// TwinCAT 3 PLC project EnOcean
// ProgramVersion: 3.1.4022.4
// libraries:
//   Tc2_BABasic, * (Beckhoff Automation GmbH)
//   Tc2_EnOcean, * (Beckhoff Automation GmbH)
//   Tc2_Standard, * (Beckhoff Automation GmbH)
//   Tc2_System, * (Beckhoff Automation GmbH)
//   Tc2_Utilities, * (Beckhoff Automation GmbH)
//   Tc3_IotBase, * (Beckhoff Automation GmbH)
//   Tc3_Module, * (Beckhoff Automation GmbH)
// project tree:
//   / GlobalTextList.TcGTLO (not stored), PlcTask.TcTTO, Visualization Manager.TcVMO (not stored)
//   GVLs/ GVL_EnOcean.TcGVL, Waardes.TcGVL
//   POUs/FB/ didSensorChange.TcPOU, isOpen.TcPOU, readTemp2.TcPOU, switch2.TcPOU, contact2.TcPOU (not stored)
//   POUs/ JSonEncode.TcPOU, Main.TcPOU, mqttconn.TcPOU, readTemp.TcPOU, switch.TcPOU, contact.TcPOU (not stored)
//   VISUs/ Visualization.TcVIS (not stored)
// real-time tasks:
//   TASK PlcTask: cycle T#5ms, priority 15, ADS port 350
// I/O:
//   DEVICE Device 1 (EtherCAT) (disabled), AmsNetId 192.168.1.6.2.1
//     Term 1 (EK1200) [EK1200-5000 EtherCAT Power supply (2A E-Bus)]
//       Term 2 (EL1008) [EL1008 8Ch. Dig. Input 24V, 3ms]
//       Term 3 (EL2008) [EL2008 8Ch. Dig. Output 24V, 0.5A]
//       Term 4 (EL3062) [EL3062 2Ch. Ana. Input 0-10V]
//       Term 5 (EL4002) [EL4002 2Ch. Ana. Output 0-10V, 12bit]
//       Box 6 (BK1250)
// variable links:
//   EnOcean/EnOcean Instance <-> Device 1 (EtherCAT)/Term 1 (EK1200)/Box 6 (BK1250)
//     PlcTask Inputs/GVL_EnOcean.stKL6581Input @bit 8 <-> Term 2 (KL6581)/Channel 1/Input CNODE
//     PlcTask Inputs/GVL_EnOcean.stKL6581Input @bit {24..48 step 8} <-> Term 2 (KL6581)/Channel 1/Input DB{0..3}  (4 links)
//     PlcTask Inputs/GVL_EnOcean.stKL6581Input @bit {56..80 step 8} <-> Term 2 (KL6581)/Channel 1/Input ID{0..3}  (4 links)
//     PlcTask Inputs/GVL_EnOcean.stKL6581Input @bit 16 <-> Term 2 (KL6581)/Channel 1/Input ORG
//     PlcTask Inputs/GVL_EnOcean.stKL6581Input @bit 88 <-> Term 2 (KL6581)/Channel 1/Input STATUS
//     PlcTask Inputs/GVL_EnOcean.stKL6581Input <-> Term 2 (KL6581)/Channel 1/Status
//     PlcTask Outputs/GVL_EnOcean.stKL6581Output <-> Term 2 (KL6581)/Channel 1/Control
//     PlcTask Outputs/GVL_EnOcean.stKL6581Output @bit 8 <-> Term 2 (KL6581)/Channel 1/Output CNODE
//     PlcTask Outputs/GVL_EnOcean.stKL6581Output @bit {24..48 step 8} <-> Term 2 (KL6581)/Channel 1/Output DB{0..3}  (4 links)
//     PlcTask Outputs/GVL_EnOcean.stKL6581Output @bit {56..80 step 8} <-> Term 2 (KL6581)/Channel 1/Output ID{0..3}  (4 links)
//     PlcTask Outputs/GVL_EnOcean.stKL6581Output @bit 16 <-> Term 2 (KL6581)/Channel 1/Output ORG
//     PlcTask Outputs/GVL_EnOcean.stKL6581Output @bit 88 <-> Term 2 (KL6581)/Channel 1/Output STATUS

CONFIGURATION EnOcean
    RESOURCE PLC ON TwinCAT3
        TASK PlcTask(INTERVAL := T#5ms, PRIORITY := 15);
        PROGRAM Main WITH PlcTask : Main;
    END_RESOURCE
END_CONFIGURATION

// ---- GVLs/GVL_EnOcean.TcGVL
{attribute 'qualified_only'}
VAR_GLOBAL
	stKL6581Input  AT %I* : KL6581_Input;
    stKL6581Output AT %Q* : KL6581_Output;
    stKL6581              : STR_KL6581;
END_VAR

// ---- GVLs/Waardes.TcGVL
{attribute 'qualified_only'}
VAR_GLOBAL
	temp 				: 	REAL;
	humitity 			: 	REAL;
	switchNR			: 	INT;
	contact1			: 	BOOL;
	contact2			:	BOOL;
	jsonHum 		    :	STRING;
	jsonTemp            :   STRING;
	jsonSwitch          :   STRING;
	Allstrings 			:   STRING(1024);
END_VAR

// ---- POUs/Main.TcPOU
PROGRAM Main
VAR
	fbKL6581			:	FB_KL6581;
	fbsearch 			:	FB_EnOcean_Search;
	//fbRecGeneric		: 	FB_Rec_Generic;
	readTemp			: 	readTemp2;
	whichSwitch			:	switch2;
	contactSensor1		: 	contact;
	contactSensor2		:	contact;
	
    temp			: 	REAL;
	humitity 			: 	REAL;
	switchNR			: 	INT;
	contact1			: 	BOOL;
	contact2			:	BOOL;
	tempError			:	BOOL;
	humitityError		: 	BOOL;
END_VAR

JsonEncode();

// Init
fbKL6581(bInit := TRUE, stKL6581_in := GVL_EnOcean.stKL6581Input, stKL6581_out := GVL_EnOcean.stKL6581Output);
GVL_EnOcean.stKL6581 := fbKL6581.str_KL6581;
fbsearch(bStart := TRUE, str_KL6581 := GVL_EnOcean.stKL6581, byNode := 0);

//link sensors aan POU
readTemp(sensorID := 92351965);
whichswitch(sensorID := 4277441636);
contactSensor1(sensorID := 84246605);
contactSensor2(sensorID := 84246605);

// IF sensor value changes
IF didSensorChange(readTemp := readTemp, whichSwitch := whichSwitch) THEN
	temp := readTemp.tempOutput;
	humitity := readTemp.humitityOut;
	switchNR := whichSwitch.switchNR;
	contact1 := contactSensor1.contact;
	contact2 := contactSensor2.contact;
	mqttconn();
END_IF
	
// handle exceptions	

IF temp < 20 OR temp > 40 THEN
	tempError := TRUE;
END_IF

IF humitity < 40 OR humitity > 60 THEN
	humitityError := TRUE;
END_IF

(*
IF switchNR <> 0 THEN
	IF switchNR = 2 THEN
		<handle switch>
	END_IF
END_IF
*)

(*
Sensor IDs:
Temp+vochtig ==> 92351965 : ar_value[1] = temp, ar_value[2] = vochtig
schakelaar ==> 4277441636 : ar_value[3]
raamcontact1 ==> 84246605 : ar_value[3]
raamcontact2 ==> 84246441: ar_value[3]




*)

END_PROGRAM

// ---- POUs/readTemp.TcPOU
PROGRAM readTemp
VAR
	fbRecGeneric		: 	FB_Rec_Generic;
END_VAR
VAR_INPUT
	sensorID			: DWORD;
END_VAR
VAR_OUTPUT
	tempOutput			: LREAL;
	humitityOut			: LREAL;
END_VAR

fbRecGeneric(str_KL6581 := GVL_EnOcean.stKL6581, byNode := 0, dw_ID := sensorID);

IF fbRecGeneric.bReceive = FALSE THEN
	tempOutput := F_Scale(fRawData := fbRecGeneric.ar_Value[1], fRawDataLowerOffLimit := 0, fRawDataUpperOffLimit := 255, fScaleDataLowerOffLimit := -20, fScaleDataUpperOffLimit := 60);
	humitityOut := F_Scale(fRawData := fbRecGeneric.ar_Value[2], fRawDataLowerOffLimit := 0, fRawDataUpperOffLimit := 255, fScaleDataLowerOffLimit := 0, fScaleDataUpperOffLimit := 100);
	
	
END_IF

END_PROGRAM

// ---- POUs/FB/readTemp2.TcPOU
FUNCTION_BLOCK readTemp2
VAR
	fbRecGeneric		: 	FB_Rec_Generic;
END_VAR
VAR_INPUT
	sensorID			: DWORD;
END_VAR
VAR_OUTPUT
	tempOutput			: LREAL;
	humitityOut			: LREAL;
END_VAR

fbRecGeneric(str_KL6581 := GVL_EnOcean.stKL6581, byNode := 0, dw_ID := sensorID);

IF fbRecGeneric.bReceive = FALSE THEN
	tempOutput := F_Scale(fRawData := fbRecGeneric.ar_Value[1], fRawDataLowerOffLimit := 0, fRawDataUpperOffLimit := 255, fScaleDataLowerOffLimit := -20, fScaleDataUpperOffLimit := 60);
	humitityOut := F_Scale(fRawData := fbRecGeneric.ar_Value[2], fRawDataLowerOffLimit := 0, fRawDataUpperOffLimit := 255, fScaleDataLowerOffLimit := 0, fScaleDataUpperOffLimit := 100);
	
	Waardes.temp := tempOutput;
	Waardes.humitity := humitityOut;
	
END_IF

END_FUNCTION_BLOCK

// ---- POUs/FB/switch2.TcPOU
FUNCTION_BLOCK switch2
VAR
	fbRecGeneric		: 	FB_Rec_Generic;
END_VAR
VAR_INPUT
	sensorID			: DWORD;
END_VAR
VAR_OUTPUT
	switchNR			: INT;
END_VAR

fbRecGeneric(str_KL6581 := GVL_EnOcean.stKL6581, byNode := 0, dw_ID := sensorID);

IF fbRecGeneric.bReceive = FALSE THEN
	IF fbRecGeneric.ar_Value[3] = 16 THEN
		switchNR := 1;
	ELSIF fbRecGeneric.ar_Value[3] = 80 THEN
		switchNR := 2;
	ELSIF fbRecGeneric.ar_Value[3] = 48 THEN
		switchNR := 3;
	ELSIF fbRecGeneric.ar_Value[3] = 112 THEN
		switchNR := 4;
	ELSE 
		switchNR := 0;
	END_IF
	Waardes.switchNR := switchNR;
END_IF

END_FUNCTION_BLOCK

// ---- POUs/JSonEncode.TcPOU
PROGRAM JSonEncode
VAR
	jsonHum  : STRING;
	jsonTemp : STRING;
	jsonSwitch : STRING;
	AllStrings: STRING(1024);
END_VAR

(*zo moet die ongeveer eruit zien
[
{"type": "sigfox", "id": "	xx	","battery": 0,"flag": 0,"mode": 0,"temp": 0,"hum": 0},

{"type": "enocean", "id": "	xx	", "value": 0},
{"type": "plc", "id": "	xx	", "raam": 0, "sprinkler": 0, "verwarming": 0}

]

 
{
    "topic": "sensordata",  <<--Deze
    "data": {
        "humidity": 0,
        "temperature": 0,
        "switch": 0
    }
}
*)
jsonHum := '';
jsonHum := concat('{"topic": "sensordata", "data": {"humidity": ', REAL_TO_STRING(waardes.humitity));
jsonHum := concat(jsonHum, ',');

Waardes.jsonHum := jsonHum;

jsonTemp := '';
jsonTemp := concat(jsonHum, '"temperature":');
jsonTemp := concat(jsonTemp, REAL_TO_STRING(waardes.temp));
jsonTemp := concat(jsonTemp, ',');

Waardes.jsonTemp := JsonTemp;

jsonSwitch := '';
jsonSwitch := concat(jsonTemp,'"switch":' );
jsonSwitch := concat(jsonSwitch, INT_TO_STRING(waardes.switchNR));
jsonSwitch := concat(jsonSwitch, '}}');

Waardes.jsonSwitch := jsonSwitch;
 
AllStrings := concat(jsonHum,JsonTemp);
AllStrings := concat(AllStrings,jsonSwitch);
Waardes.Allstrings := Allstrings;

END_PROGRAM

// ---- POUs/switch.TcPOU
PROGRAM switch
VAR
	fbRecGeneric		: 	FB_Rec_Generic;
END_VAR
VAR_INPUT
	sensorID			: DWORD;
END_VAR
VAR_OUTPUT
	switchNR			: INT;
END_VAR

fbRecGeneric(str_KL6581 := GVL_EnOcean.stKL6581, byNode := 0, dw_ID := sensorID);

IF fbRecGeneric.bReceive = FALSE THEN
	IF fbRecGeneric.ar_Value[3] = 16 THEN
		switchNR := 1;
	ELSIF fbRecGeneric.ar_Value[3] = 80 THEN
		switchNR := 2;
	ELSIF fbRecGeneric.ar_Value[3] = 96 THEN
		switchNR := 3;
	ELSIF fbRecGeneric.ar_Value[3] = 112 THEN
		switchNR := 4;
	ELSE 
		switchNR := 0;
	END_IF
END_IF

END_PROGRAM

// ---- POUs/FB/didSensorChange.TcPOU
FUNCTION didSensorChange : BOOL
VAR_INPUT
	readTemp			: 	readTemp2;
	whichSwitch			:	switch2;
END_VAR
VAR
END_VAR

IF readTemp.fbRecGeneric.bReceive = FALSE OR whichSwitch.fbRecGeneric.bReceive = FALSE THEN
	didSensorChange := TRUE;
	ELSE
		didSensorChange := FALSE;
END_IF

END_FUNCTION

// ---- POUs/mqttconn.TcPOU
PROGRAM mqttconn
VAR
    fbMqttClient    : FB_IotMqttClient;
	
    bSetParameter   : BOOL := TRUE;
    bConnect        : BOOL := TRUE;

	    (* published message *)
    sTopicPub   : STRING(255) := 'test'; //test/message (rabbitmq, pi)
    sPayloadPub : STRING(255);
    i : UDINT;
    fbTimer : TON := (PT:=T#1S);

    (* received message *)
    bSubscribed    : BOOL;
    sTopicSub      : STRING(255) := 'test';
    {attribute 'TcEncoding':='UTF-8'}
    sTopicRcv      : STRING(255);
    {attribute 'TcEncoding':='UTF-8'}
    sPayloadRcv    : STRING(255);
    fbMessageQueue : FB_IotMqttMessageQueue;
    fbMessage      : FB_IotMqttMessage;
	
	redge : r_trig;
	bexec : bool;
END_VAR

IF bSetParameter THEN
    bSetParameter               := FALSE;
    fbMqttClient.sHostName      := '192.168.1.175';
    fbMqttClient.nHostPort      := 1883;
//fbMqttClient.sClientId      := ''; 
    fbMqttClient.sTopicPrefix   := ''; 
    fbMqttClient.nKeepAlive     := 60; 
    //fbMqttClient.sUserName      := 'admin' ;
   // fbMqttClient.sUserPassword  := 'password'; 
//  fbMqttClient.stWill         := ; 
//  fbMqttClient.stTLS          := ;
    fbMqttClient.ipMessageQueue := fbMessageQueue;
END_IF
fbMqttClient.Execute(bConnect);

IF fbMqttClient.bConnected THEN
    IF NOT bSubscribed THEN
        bSubscribed := fbMqttClient.Subscribe(sTopic:=sTopicSub, eQoS:=TcIotMqttQos.AtMostOnceDelivery);
    END_IF
    fbTimer(IN:=TRUE);
    IF fbTimer.Q THEN // publish new payload every second
        fbTimer(IN:=FALSE);
        i := i + 1;
        //sPayloadPub := CONCAT('test number is ', TO_STRING(i));
		sPayloadPub := Waardes.Allstrings;
        fbMqttClient.Publish(    sTopic:= sTopicPub, 
                                pPayload:= ADR(sPayloadPub), nPayloadSize:= LEN2(ADR(sPayloadPub))+1, 
                                eQoS:= TcIotMqttQos.AtMostOnceDelivery, bRetain:= FALSE, bQueue:= FALSE );
    END_IF
END_IF

IF fbMessageQueue.nQueuedMessages > 0 THEN
    IF fbMessageQueue.Dequeue(fbMessage:=fbMessage) THEN
        fbMessage.GetTopic(pTopic:=ADR(sTopicRcv), nTopicSize:=SIZEOF(sTopicRcv) );
        fbMessage.GetPayload(pPayload:=ADR(sPayloadRcv), nPayloadSize:=SIZEOF(sPayloadRcv), bSetNullTermination:=FALSE);
    END_IF
END_IF

redge(clk := bexec);

IF(redge.Q)THEN
	i := i + 1;
        sPayloadPub := CONCAT('test number is ', TO_STRING(i));
        fbMqttClient.Publish(    sTopic:= sTopicPub, 
                                pPayload:= ADR(sPayloadPub), nPayloadSize:= LEN2(ADR(sPayloadPub))+1, 
                                eQoS:= TcIotMqttQos.AtMostOnceDelivery, bRetain:= FALSE, bQueue:= FALSE );
	bexec := FALSE;
	
END_IF

END_PROGRAM

// ---- POUs/FB/isOpen.TcPOU
FUNCTION isOpen : BOOL
VAR_INPUT
	sensorID			:	DWORD;
END_VAR
VAR
	fbRecGeneric		: 	FB_Rec_Generic;
END_VAR

fbRecGeneric(str_KL6581 := GVL_EnOcean.stKL6581, byNode := 0, dw_ID := sensorID);

IF fbRecGeneric.ar_Value[3] = 8 THEN
	isOpen := TRUE;
ELSE
	isOpen := FALSE;
END_IF

END_FUNCTION
